FUNCTION_BLOCK FB_Leica
VAR_INPUT
END_VAR
VAR_OUTPUT
	// Leica Variables
	AngleHz			AT %I* : LREAL := 0.0;
	AngleVt			AT %I* : LREAL := 0.0;
	Distance		AT %I* : LREAL := 0.0;
	q0				AT %I* : LREAL := 0.0;
	q1				AT %I* : LREAL := 0.0;
	q2				AT %I* : LREAL := 0.0;
	q3				AT %I* : LREAL := 0.0;
	TimeStamp		AT %I* : ULINT := 0;
	
	x				: LREAL := 0.0;
	y				: LREAL := 0.0;
	z				: LREAL := 0.0;
END_VAR
VAR
	
	
	
END_VAR

// Leica transform to x,y and z coordinates
x := Distance*SIN(AngleVt)*SIN(AngleHz);
y := Distance*SIN(AngleVt)*COS(AngleHz);
z := Distance*COS(AngleVt);

END_FUNCTION_BLOCK

(* stored: Version 1.1.0.1, ProductVersion 3.1.4020.12
   POU FB_Leica: Id {b81552ff-c250-4296-8f9a-58288f81cd30}, SpecialFunc None *)
